// TIA Portal project "Projekt1500" (V17)

(* hardware
DEVICE "S7-1500/ET200MP-Station_1"  S7-1500 station
   slot 0: "Profilschiene_0"  Rack  6ES7 590-1***0-0AA0
   slot 1: "PLC_1"  CPU 1516-3 PN/DP  6ES7 516-3AN00-0AB0  V1.8
      slot 3: "CPU-Display_1"  6ES7591-1BA00-0AA0
      slot 32768: "PROFINET-Schnittstelle_1"  X1
         slot 32769: "Port_1"  X1 P1
         slot 32770: "Port_2"  X1 P2
      slot 33024: "PROFINET-Schnittstelle_2"  X2
         slot 33025: "Port_1"  X2 P1
      slot 33280: "DP-Schnittstelle_1"  X3
   slot 2: "DQ 32x24VDC/0.5A BA_1"  DQ 32x24VDC/0.5A BA  6ES7 522-1BL10-0AA0  V1.1
   slot 3: "DI 32x24VDC BA_1"  DI 32x24VDC BA  6ES7 521-1BL10-0AA0  V1.1
*)

// ===== PLC "PLC_1"  CPU 1516-3 PN/DP =====

VAR_GLOBAL   // PLC tag table "Standard-Variablentabelle"
   "P1" AT %Q0.0 : Bool;   // Meldeleuchte
   "System_Byte" AT %MB100 : Byte;
   "FirstScan" AT %M100.0 : Bool;
   "DiagStatusUpdate" AT %M100.1 : Bool;
   "AlwaysTRUE" AT %M100.2 : Bool;
   "AlwaysFALSE" AT %M100.3 : Bool;
   "Clock_Byte" AT %MB110 : Byte;
   "Clock_10Hz" AT %M110.0 : Bool;
   "Clock_5Hz" AT %M110.1 : Bool;
   "Clock_2.5Hz" AT %M110.2 : Bool;
   "Clock_2Hz" AT %M110.3 : Bool;
   "Clock_1.25Hz" AT %M110.4 : Bool;
   "Clock_1Hz" AT %M110.5 : Bool;
   "Clock_0.625Hz" AT %M110.6 : Bool;
   "Clock_0.5Hz" AT %M110.7 : Bool;
   "S1" AT %I0.0 : Bool;   // Taster Start
END_VAR

DATA_BLOCK "PcToPlc"   // DB1
{ S7_Optimized_Access := 'FALSE' }
VERSION : 0.1
   VAR
      Plc : Array[0..256] of Byte;
   END_VAR
BEGIN
END_DATA_BLOCK

DATA_BLOCK "PlcToPc"   // DB2
{ S7_Optimized_Access := 'FALSE' }
VERSION : 0.1
   VAR
      Plc : Array[0..256] of Byte;
   END_VAR
BEGIN
END_DATA_BLOCK

DATA_BLOCK "DeleteMe_DB"   // DB3
{ S7_Optimized_Access := 'TRUE' }
VERSION : 0.1
// stored: InstanceOfName DeleteMe
"DeleteMe"
BEGIN
END_DATA_BLOCK

FUNCTION_BLOCK "DeleteMe"   // FB1, SCL
{ S7_Optimized_Access := 'TRUE' }
VERSION : 0.1
   VAR
      Eingeschaltet : Bool;
      Gesamtzeit : TON_TIME;
   END_VAR
BEGIN
END_FUNCTION_BLOCK

FUNCTION "DatenRangieren" : Void   // FC1, SCL
{ S7_Optimized_Access := 'TRUE' }
VERSION : 0.1
   VAR_TEMP
      TextLaenge : UInt;
   END_VAR
BEGIN
   // Area 16#81 --> Input
   // Area 16#82 --> Output
   // Area 16#84 --> DB

   IF  "PcToPlc".Plc[96].%X0 THEN
       // Simulation aktiv --> DI werden vom PC überschrieben
       POKE(area := 16#81,                     // DI (Hardware PLC)
           dbNumber := 0,
           byteOffset := 0,
           value := PEEK(area := 16#84, dbNumber := 1, byteOffset := 0));
   ELSE
       // Hardware aktiv --> DI werden zum PC übertragen
       POKE(area := 16#84,                    // Datenbausteine
           dbNumber := 1,                     // DB1 -> Pc2Plc
           byteOffset := 0,                   // Byte 0
           value := PEEK(area := 16#81, dbNumber := 0, byteOffset := 0));
   END_IF;

   // DQ werden immer zum PC übertragen
   POKE(area := 16#84,                         // Datenbausteine
        dbNumber := 2,                         // DB1 -> Pc2Plc
        byteOffset := 0,
        value := PEEK(area := 16#82, dbNumber := 0, byteOffset := 0));

   Strg_TO_Chars(Strg := 'Fibonacci V3.0',
                 pChars := 96,
                 Cnt=>#TextLaenge,
                 Chars := "PlcToPc".Plc);
END_FUNCTION

ORGANIZATION_BLOCK "Main"   // OB1, LAD, ProgramCycle
TITLE = "Main Program Sweep (Cycle)"
{ S7_Optimized_Access := 'TRUE' }
VERSION : 0.1
   VAR_INPUT
      Initial_Call : Bool;   // Initial call of this OB
      Remanence : Bool;   // =True, if remanent data are available
   END_VAR
BEGIN

REGION Network 1
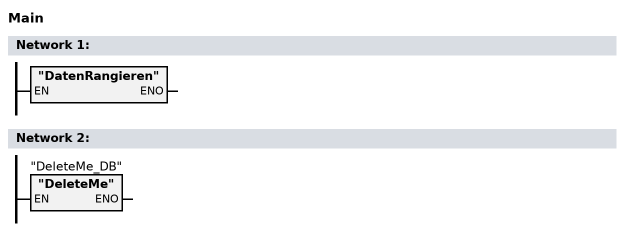
   RUNG wire#powerrail
      "DatenRangieren"()
   END_RUNG
   // the same network as SCL:
   "DatenRangieren"();
END_REGION

REGION Network 2
   RUNG wire#powerrail
      "DeleteMe_DB"()
   END_RUNG
   // the same network as SCL:
   "DeleteMe_DB"();   // "DeleteMe"
END_REGION
END_ORGANIZATION_BLOCK

ORGANIZATION_BLOCK "Startup"   // OB100, SCL, Startup
TITLE = "Complete Restart"
{ S7_Optimized_Access := 'TRUE' }
VERSION : 0.1
   VAR_INPUT
      LostRetentive : Bool;   // True if retentive data are lost
      LostRTC : Bool;   // True if date and time are lost
   END_VAR
BEGIN
   // Area 16#81 --> Input
   // Area 16#82 --> Output
   // Area 16#84 --> DB

   POKE(area := 16#82, dbNumber := 0, byteOffset := 0, value := byte#0);  // Ausgänge löschen
END_ORGANIZATION_BLOCK